// TIA Portal V18 export
// export: Created 2025-12-01T17:51:07.5454431Z, ExportSetting None, DisplayName Totally Integrated Automation Portal, DisplayVersion V18 Update 5, DisplayName TIA Portal Openness, DisplayVersion V18 Update 5, DisplayName TIA Portal Teamcenter Gateway, DisplayVersion V18, DisplayName TIA Portal Version Control Interface, DisplayVersion V18, DisplayName STEP 7 Professional, DisplayVersion V18 Update 5, DisplayName STEP 7 Safety, DisplayVersion V18, DisplayName WinCC Professional, DisplayVersion V18 Update 5
DATA_BLOCK "ST10_SafetyGate6_DB"   // DB1146
// stored: AutoNumber false, InstanceOfName SafetyGate, InstanceOfType FB
"SafetyGate"
   // VAR_INPUT
   //    iSysInface : "RCS_SysComInterface_V1";
   //    "iSafetyGate Opened Monitor" : Bool;
   //    "iSafetyGate Locked Monitor" : Bool;
   //    i1s_Pulse : Bool;
   //    "iSafetyGate AutoLock Timer" : Time;
   //    "iSafetyGate ManualLock Timer" : Time;
   //    iMode : Int;
   // END_VAR
   // VAR_OUTPUT
   //    "oSafetyGate LockedLamp" { ExternalAccessible := 'False'; ExternalVisible := 'False'; ExternalWritable := 'False'} : Bool;
   // END_VAR
   // VAR_IN_OUT
   //    ioSafetyGateLock : Bool;
   //    ioHMI_Interface : "SafetyGateUDT";
   // END_VAR
   // VAR
   //    "sSafetyGate Timer" { S7_SetPoint := 'True'} : Array[1..5] of TON_TIME;
   //    sP_Trig : Array[1..10] of Bool;
   //    sN_Trig : Array[1..10] of Bool;
   //    "sSafetyGate UnlockRequest" { ExternalAccessible := 'False'; ExternalVisible := 'False'; ExternalWritable := 'False'} : Bool;
   //    "sSafetyGate LockRequest" : Bool;
   // END_VAR
BEGIN
END_DATA_BLOCK
